TYPE NET_VAR_DATA :
STRUCT
	CYCLE : UDINT;
	STATE : BYTE;
	INDEX : INT;
	ID_MAX : USINT;
	ERROR_ID : BYTE;
	BUF_SIZE : UINT;
	S_BUF : NETWORK_BUFFER;
	R_BUF : NETWORK_BUFFER;
END_STRUCT
END_TYPE

(* stored: Version 1.1.0.1, ProductVersion 3.1.4022.7
   DUT NET_VAR_DATA: Id {17b36d3b-e584-4980-b8d7-b728389cec02} *)
